Staubli VAL3: oCryoLongOut.pgx

public program oCryoLongOut(num nChoice (dimensions=1))
// oCryoLongOut
begin
  dioSet(oCryoLongOut,nChoice)
end
